Staubli VAL3: insertItem.pgx

public program insertItem(num x_nIndexCopy, num x_nIndexPaste)
  local num l_nLastType
  local point l_pPoint
  local num l_nType
  local joint l_jJoint
begin
  //
  // use to add more elements from the typical one
  //
  // insert all the field
  //
  // JOINT
  l_jJoint=jEditPoint.tData[x_nIndexCopy].jJoint
  insert(jEditPoint.tData[x_nIndexPaste])
  jEditPoint.tData[x_nIndexPaste].jJoint=l_jJoint

end
